// TIA Portal V16 export
// export: Created 2021-03-04T22:04:03.7428455Z, ExportSetting WithDefaults, DisplayName Totally Integrated Automation Portal, DisplayVersion V16, DisplayName TIA Portal Version Control Interface, DisplayVersion V16, DisplayName TIA Portal Openness, DisplayVersion V16, DisplayName SINAMICS Startdrive Advanced, DisplayVersion V16, DisplayName SINAMICS Startdrive G130, G150, S120, S150, SINAMICS MV, S210, DisplayVersion V16, DisplayName SINAMICS Startdrive G110M, G120, G120C, G120D, G120P, DisplayVersion V16, DisplayName STEP 7 Professional, DisplayVersion V16, DisplayName STEP 7 Safety, DisplayVersion V16, DisplayName WinCC Professional, DisplayVersion V16
FUNCTION "fcBitsToWord" : Void   // FC301, LAD
TITLE = Pack Bits into word
{ S7_Optimized_Access := 'TRUE' }
AUTHOR : DMC
FAMILY : LowLevel
VERSION : 0.1
// stored: AutoNumber false, IsIECCheckEnabled false, SetENOAutomatically false, UDAEnableTagReadback false
   VAR_INPUT
      bInBit00 : Bool;   // Bit 0
      bInBit01 : Bool;   // Bit 1
      bInBit02 : Bool;   // Bit 2
      bInBit03 : Bool;   // Bit 3
      bInBit04 : Bool;   // Bit 4
      bInBit05 : Bool;   // Bit 5
      bInBit06 : Bool;   // Bit 6
      bInBit07 : Bool;   // Bit 7
      bInBit08 : Bool;   // Bit 8
      bInBit09 : Bool;   // Bit 9
      bInBit10 : Bool;   // Bit 10
      bInBit11 : Bool;   // Bit 11
      bInBit12 : Bool;   // Bit 12
      bInBit13 : Bool;   // Bit 13
      bInBit14 : Bool;   // Bit 14
      bInBit15 : Bool;   // Bit 15
   END_VAR
   VAR_OUTPUT
      wOutWord : Word;   // Packed Word
   END_VAR
BEGIN

REGION Network 1: Bit0
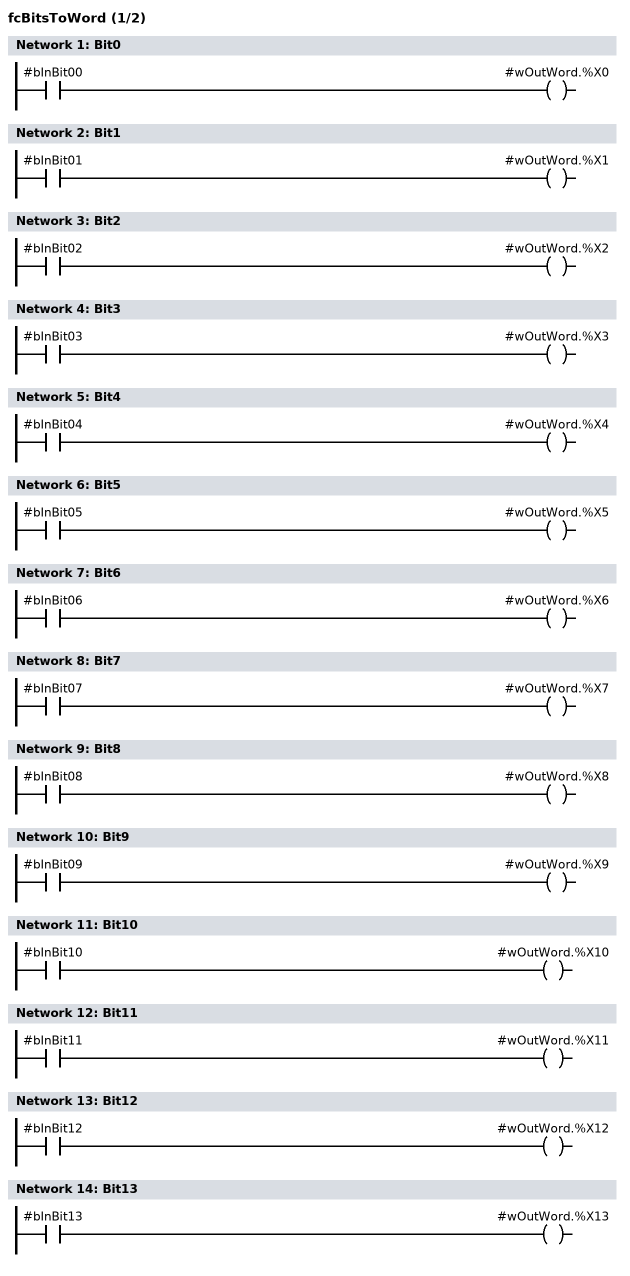
   RUNG wire#powerrail
      Contact( #bInBit00 )
      Coil( #wOutWord.%X0 )
   END_RUNG
   // the same network as SCL:
   #wOutWord.%X0 := #bInBit00;
END_REGION

REGION Network 2: Bit1
   RUNG wire#powerrail
      Contact( #bInBit01 )
      Coil( #wOutWord.%X1 )
   END_RUNG
   // the same network as SCL:
   #wOutWord.%X1 := #bInBit01;
END_REGION

REGION Network 3: Bit2
   RUNG wire#powerrail
      Contact( #bInBit02 )
      Coil( #wOutWord.%X2 )
   END_RUNG
   // the same network as SCL:
   #wOutWord.%X2 := #bInBit02;
END_REGION

REGION Network 4: Bit3
   RUNG wire#powerrail
      Contact( #bInBit03 )
      Coil( #wOutWord.%X3 )
   END_RUNG
   // the same network as SCL:
   #wOutWord.%X3 := #bInBit03;
END_REGION

REGION Network 5: Bit4
   RUNG wire#powerrail
      Contact( #bInBit04 )
      Coil( #wOutWord.%X4 )
   END_RUNG
   // the same network as SCL:
   #wOutWord.%X4 := #bInBit04;
END_REGION

REGION Network 6: Bit5
   RUNG wire#powerrail
      Contact( #bInBit05 )
      Coil( #wOutWord.%X5 )
   END_RUNG
   // the same network as SCL:
   #wOutWord.%X5 := #bInBit05;
END_REGION

REGION Network 7: Bit6
   RUNG wire#powerrail
      Contact( #bInBit06 )
      Coil( #wOutWord.%X6 )
   END_RUNG
   // the same network as SCL:
   #wOutWord.%X6 := #bInBit06;
END_REGION

REGION Network 8: Bit7
   RUNG wire#powerrail
      Contact( #bInBit07 )
      Coil( #wOutWord.%X7 )
   END_RUNG
   // the same network as SCL:
   #wOutWord.%X7 := #bInBit07;
END_REGION

REGION Network 9: Bit8
   RUNG wire#powerrail
      Contact( #bInBit08 )
      Coil( #wOutWord.%X8 )
   END_RUNG
   // the same network as SCL:
   #wOutWord.%X8 := #bInBit08;
END_REGION

REGION Network 10: Bit9
   RUNG wire#powerrail
      Contact( #bInBit09 )
      Coil( #wOutWord.%X9 )
   END_RUNG
   // the same network as SCL:
   #wOutWord.%X9 := #bInBit09;
END_REGION

REGION Network 11: Bit10
   RUNG wire#powerrail
      Contact( #bInBit10 )
      Coil( #wOutWord.%X10 )
   END_RUNG
   // the same network as SCL:
   #wOutWord.%X10 := #bInBit10;
END_REGION

REGION Network 12: Bit11
   RUNG wire#powerrail
      Contact( #bInBit11 )
      Coil( #wOutWord.%X11 )
   END_RUNG
   // the same network as SCL:
   #wOutWord.%X11 := #bInBit11;
END_REGION

REGION Network 13: Bit12
   RUNG wire#powerrail
      Contact( #bInBit12 )
      Coil( #wOutWord.%X12 )
   END_RUNG
   // the same network as SCL:
   #wOutWord.%X12 := #bInBit12;
END_REGION

REGION Network 14: Bit13
   RUNG wire#powerrail
      Contact( #bInBit13 )
      Coil( #wOutWord.%X13 )
   END_RUNG
   // the same network as SCL:
   #wOutWord.%X13 := #bInBit13;
END_REGION

REGION Network 15: Bit14
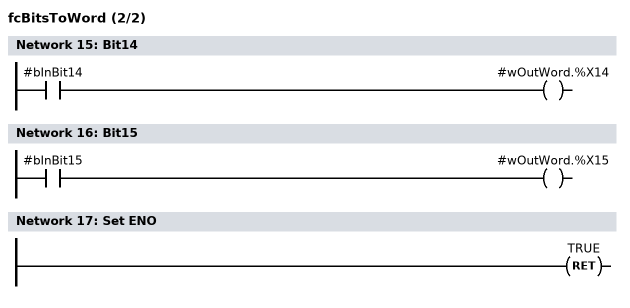
   RUNG wire#powerrail
      Contact( #bInBit14 )
      Coil( #wOutWord.%X14 )
   END_RUNG
   // the same network as SCL:
   #wOutWord.%X14 := #bInBit14;
END_REGION

REGION Network 16: Bit15
   RUNG wire#powerrail
      Contact( #bInBit15 )
      Coil( #wOutWord.%X15 )
   END_RUNG
   // the same network as SCL:
   #wOutWord.%X15 := #bInBit15;
END_REGION

REGION Network 17: Set ENO
   RUNG wire#powerrail
      ReturnCoil( TRUE )
   END_RUNG
   // the same network as SCL:
   ENO := TRUE;
   RETURN;
END_REGION
END_FUNCTION
